//==================================================================================================
//							Beckhoff Automation Poland
//									24.04.2018
//	Struktura zawierajaca najwazniejsze statusy osi
//  v1.0	|| TC v 3.1.4022.16		|| - pierwsza wersja
//==================================================================================================
TYPE ST_McAxisStatus :
STRUCT
	stAxisStatus			: Tc2_MC2.ST_AxisStatus;
	sAxisName				: STRING(31);				// 
	dwAxisId				: DWORD;					// Axis ID
	bNcError				: BOOL;						// Nc Eror flag
	udiNcErrorCode			: UDINT;					// Nc axis error code
	{attribute 'displaymode':='hex'}
	udiNcErrorCodeHex		: UDINT;					// Nc axis error code - hex format
	lrActPos				: LREAL;					// Actual position (absolut value from NC)
	lrModuloActPos			: LREAL;					// Actual modulo position (absolut value from NC)
	lrActVelo				: LREAL;					// Actual velocity
	lrActAcc				: LREAL;					// Actual acceleration
	lrActTorque				: LREAL;
	lrSetPos				: LREAL;					// Set position (absolut value from NC)
	lrSetVelo				: LREAL;					// Set velocity
	lrSetAcc				: LREAL;					// Set acceleration
	lrSetTorque				: LREAL;

	lrPosDiff				: LREAL;					// Position difference (lag distance)
	bAxisReady				: BOOL;						// Axis.Status.Operational
	bHomed					: BOOL;
	bCoupled				: BOOL;
	bAcceptBlockedDrive		: BOOL;						// Force move back from limit switch
END_STRUCT
END_TYPE

(* stored: Version 1.1.0.1, ProductVersion 3.1.4026.13, FileIdentifier 13b832b809f66d23a1a7c3446c9792a0a30db8ae, FileSignature 952875e4bbed1f20a110ca5d2a82ce2a34776854a2f765ad07d0a4771b363e3ba538540dd369c4efd4ebeb631138fd2ae3e7b4c4e854f370aed4feacba3be811a02025c0fa16605c9d2327f255886c3432068d226782a890d08b5210c7ffca97cc0fb1ac95c83ff3ab472888eaeb1dfc1ada40ac7e7f88d2a226561a9074bedc66afbc59ff74a739c9c07ae37bd54277ed2f9624e1002dacb9f65bce16a3c426420883027ab96fc98fa9e3818fd3962808641cfb1e9c38ee3c572678e59b8451cc17412a1e31d7f674a4682bdc262bf7d86fc6f1e7a2849e99c4b7570956ccb507d4b42d9f21a1cba346608c4c8199aab873134aab13b309529b7af0eef0db4f
   DUT ST_McAxisStatus: Id {fc3ec117-11de-47a7-867d-a0d2bfeacbec} *)
